Staubli VAL3: getPosition.pgx

program getPosition(string getCommandName, joint requestedJoint, num sio_ID)
  local string message
  local pointRx readPosition
begin
  //**************************************************
  // Returns the contents of the trsf of the requested position.
  // On testing, we found that whereas a distance can be requested with
  // 2 or 3dp of precision, angles could not (got a runtime error on
  // the robot. Hence we return angles with no dp; we only need 2dp for
  // distances.
  //**************************************************
  putln("getPosition:")
  putln("   "+getCommandName)
  readPosition=jointToPoint(flange,world,requestedJoint)
  message=getCommandName+":#X"+toString(".2",readPosition.trsf.x)
  message=message+"#Y"+toString(".2",readPosition.trsf.y)
  message=message+"#Z"+toString(".2",readPosition.trsf.z)
  message=message+"#RX"+toString("",readPosition.trsf.rx)
  message=message+"#RY"+toString("",readPosition.trsf.ry)
  message=message+"#RZ"+toString("",readPosition.trsf.rz)

  call sendStatus(message,sio_ID)
end
